PROGRAM MAIN
VAR
	fbStepWorker : FB_StepWorker;
	Valve1 : Actuator;
	Valve2 : Actuator;
	Valve3 : Actuator;
	fbUintComparator : UintComparator;
	uiCounter : UINT;
	uiDesiredStep : UINT := 10;
	fbRelease : Boolean;
	bReportTimeout : BOOL;
	test : BOOLIN;
	test2 : BOOLIN;
	sAppName : STRING;
	sProjectName : STRING;
	SystemInfo : PlcAppSystemInfo;
	SymbolPathStorage : SymbolPathStorage;
END_VAR

SystemInfo := _AppInfo;
sAppName := _AppInfo.AppName;
sProjectName := _AppInfo.ProjectName; 

fbUintComparator();
fbStepWorker();

CASE fbStepWorker.uiStep OF

	0:	
	
		fbUintComparator.mEquals(fbStepWorker.uiStep,uiDesiredStep);
		
		fbStepWorker
			.mAddCondition(Valve1.fbOutput)
			.mAddCondition(Valve2.fbOutput)
			.mAddCondition(Valve3.fbOutput);
			
		fbStepWorker.mNextStep(10);
		
		
	10:	
	
		fbStepWorker
			.mSetTimeout(T#10S)
			.mAddCondition(fbUintComparator)
			.mAddCondition(fbRelease);
			
		fbStepWorker.mNextStep(20);
		bReportTimeout := fbStepWorker.bTimeout;
		
	20:
		;
	
END_CASE;

END_PROGRAM

(* stored: Version 1.1.0.1, ProductVersion 3.1.4024.2
   POU MAIN: Id {b63b2f9e-7008-4ed9-b68d-d2eaed7795ed}, SpecialFunc None *)
